(* Logix 5000 project; controller R5_CSS vendor 1 type 14 code 74 rev 19.11; software revision 19.01; part 16 of 20 *)
(* tags used below, declared in another part *)
   AlarmMaster : DINT;
   AllowHeatersWhenEmpty : BOOL;
   FT140_TOTAL_FLOW : REAL;
   HT_FAULT : BOOL;
   LC303B : LEVEL_CONTROL;   // INTERFACE LEVEL OF PRIMARY CONDENSER
   MV115B : ValveControl_TwoWay;
   MV301 : ValveControl_TwoWay;
   option_CartridgeHeaters : BOOL;
   P101A : PUMP_CONTROL;
   P101B : PUMP_CONTROL;
   P302A : PUMP_CONTROL;
   P302B : PUMP_CONTROL;
   P305 : PUMP_CONTROL;
   PID_JHE102 : PID;
   PID_JHE102_TON : TIMER;
   PID_TCV108 : PID;   // QUENCH FEED CONTROL VALVE
   PID_TCV108_Flow : PID;
   PID_TCV108_TON : TIMER;
   QuenchFlowMeterFailed : BOOL;
   QuenchTowerControlMode : BOOL;   // 0 = Temp.control 1 = Flow control
   TC101A : TEMP_CONTROL;   // QUENCH BASIN TRANSFER BASIN A TEMPERATURE CONTROL
   TC101B : TEMP_CONTROL;   // QUENCH BASIN TRANSFER BASIN B TEMPERATURE CONTROL
   TC108 : TEMP_CONTROL;   // QUENCH TOWER EXIT GAS TEMPERATURE CONTROL
   TC108_AUTO_ONS1 : BOOL;
   TC108_AUTO_ONS2 : BOOL;
   TC108_AutoStatic_SeekMaxSec : DINT;
   TC108_AutoStatic_SeekMaxTime : BOOL;
   TC108_AutoStatic_SeekMaxTmr : TIMER;
   TC108_AutoStatic_SeekTmr : TIMER;
   TC108_AutoStatic_SP : REAL;
   TC108_AutoStatic_SP_DB : REAL;
   TC108_AutoStatic_SP_DB_Down : REAL;
   TC108_AutoStatic_SP_DB_Up : REAL;
   TC108_manual_ONS1 : BOOL;
   TC108_QuenchFlowMeterFailedHold : REAL;
   TC108_QuenchFlowMeterFailedONS : BOOL;
   TC108_StaticMode : BOOL;
   TC108_StaticMode_Seek : BOOL;
   TC112 : TEMP_CONTROL;   // Quench Water Cartridge Heater ProcessTemp
   TC112_AUTO_Ons : BOOL;
   TC112_AUTO_Ons1 : BOOL;
   TC112_HeaterDisabled : BOOL;
   TC112_MANUAL_Ons : BOOL;
   TC112_NoPumpsRunningAlm : BOOL;
   TC112_START_TON : TIMER;
   TC112A : TEMP_CONTROL;
   TC313B : TEMP_CONTROL;   // PRIMARY COALESCER SHELL TEMPERATURE CONTROL
   TC319 : TEMP_CONTROL;   // COALESCER OIL CHAMBER PROCESS TEMPERATURE CONTROL
   TC319A : TEMP_CONTROL;   // COALESCER OIL CHAMBER SHEATH TEMPERATURE
   TMR_FAULT : DINT;
(* MainProgram, continued *)

ROUTINE TC101A_BasinPumpTemperature   (* ladder *)
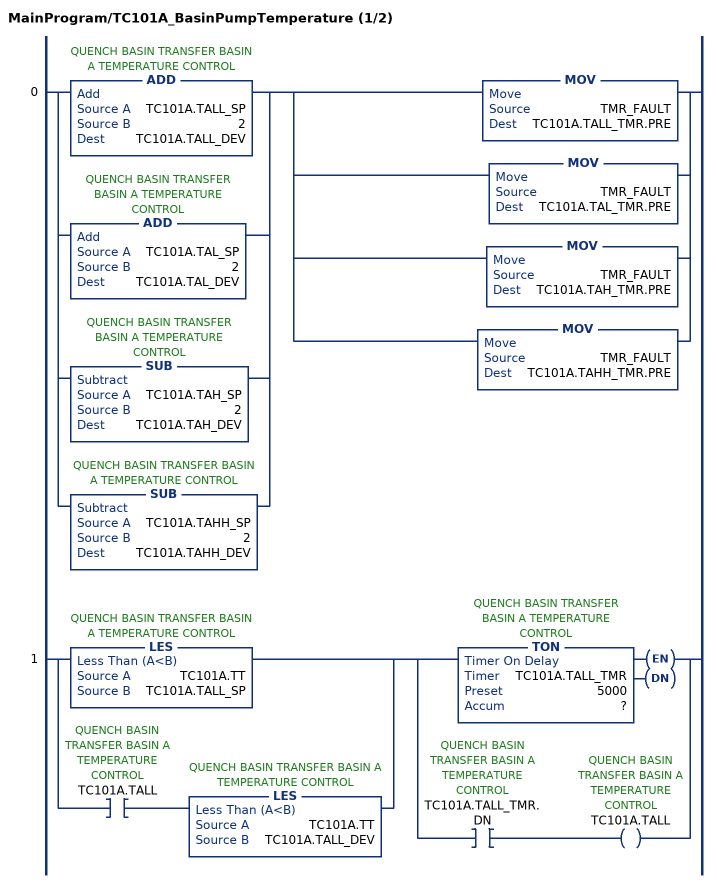
   0: [ADD(TC101A.TALL_SP,2,TC101A.TALL_DEV) ,ADD(TC101A.TAL_SP,2,TC101A.TAL_DEV) ,SUB(TC101A.TAH_SP,2,TC101A.TAH_DEV) ,SUB(TC101A.TAHH_SP,2,TC101A.TAHH_DEV) ][MOV(TMR_FAULT,TC101A.TALL_TMR.PRE) ,MOV(TMR_FAULT,TC101A.TAL_TMR.PRE) ,MOV(TMR_FAULT,TC101A.TAH_TMR.PRE) ,MOV(TMR_FAULT,TC101A.TAHH_TMR.PRE) ];
   1: [LES(TC101A.TT,TC101A.TALL_SP) ,XIC(TC101A.TALL) LES(TC101A.TT,TC101A.TALL_DEV) ][TON(TC101A.TALL_TMR,?,?) ,XIC(TC101A.TALL_TMR.DN) OTE(TC101A.TALL) ];
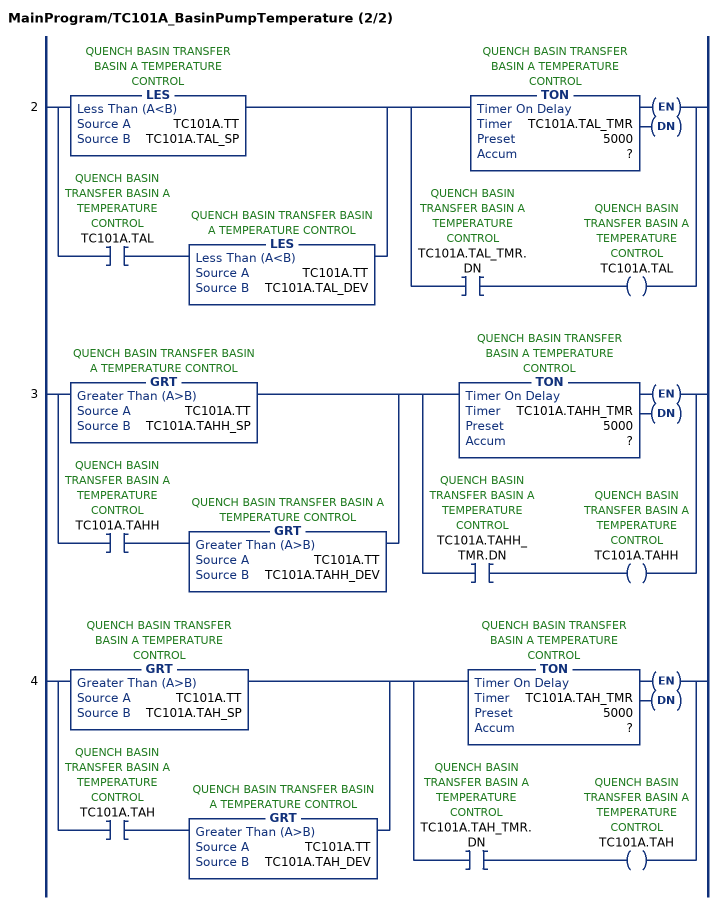
   2: [LES(TC101A.TT,TC101A.TAL_SP) ,XIC(TC101A.TAL) LES(TC101A.TT,TC101A.TAL_DEV) ][TON(TC101A.TAL_TMR,?,?) ,XIC(TC101A.TAL_TMR.DN) OTE(TC101A.TAL) ];
   3: [GRT(TC101A.TT,TC101A.TAHH_SP) ,XIC(TC101A.TAHH) GRT(TC101A.TT,TC101A.TAHH_DEV) ][TON(TC101A.TAHH_TMR,?,?) ,XIC(TC101A.TAHH_TMR.DN) OTE(TC101A.TAHH) ];
   4: [GRT(TC101A.TT,TC101A.TAH_SP) ,XIC(TC101A.TAH) GRT(TC101A.TT,TC101A.TAH_DEV) ][TON(TC101A.TAH_TMR,?,?) ,XIC(TC101A.TAH_TMR.DN) OTE(TC101A.TAH) ];
END_ROUTINE

ROUTINE TC101B_BasinPumpTemperature   (* ladder *)
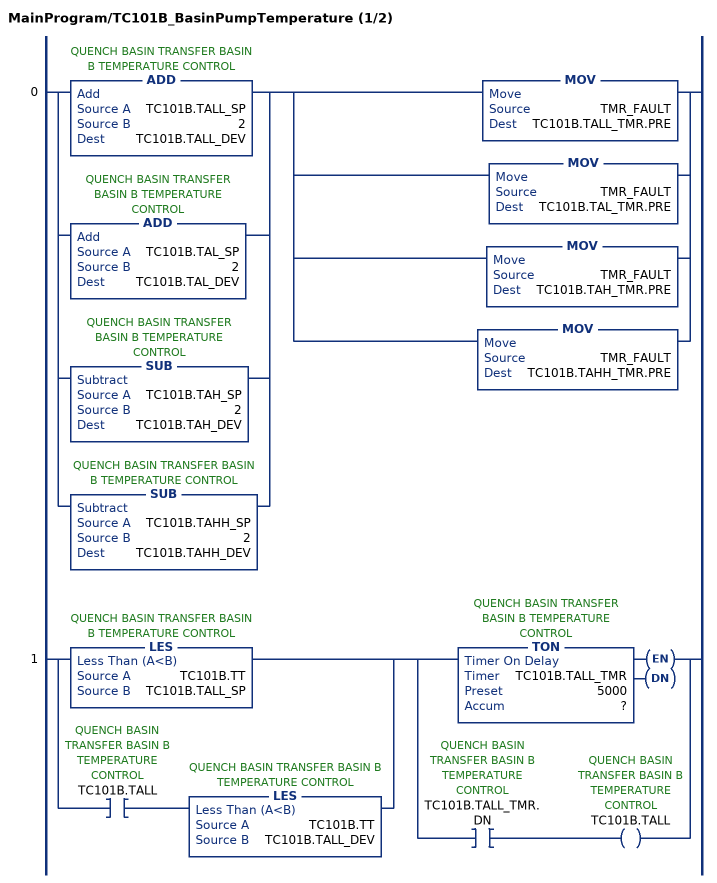
   0: [ADD(TC101B.TALL_SP,2,TC101B.TALL_DEV) ,ADD(TC101B.TAL_SP,2,TC101B.TAL_DEV) ,SUB(TC101B.TAH_SP,2,TC101B.TAH_DEV) ,SUB(TC101B.TAHH_SP,2,TC101B.TAHH_DEV) ][MOV(TMR_FAULT,TC101B.TALL_TMR.PRE) ,MOV(TMR_FAULT,TC101B.TAL_TMR.PRE) ,MOV(TMR_FAULT,TC101B.TAH_TMR.PRE) ,MOV(TMR_FAULT,TC101B.TAHH_TMR.PRE) ];
   1: [LES(TC101B.TT,TC101B.TALL_SP) ,XIC(TC101B.TALL) LES(TC101B.TT,TC101B.TALL_DEV) ][TON(TC101B.TALL_TMR,?,?) ,XIC(TC101B.TALL_TMR.DN) OTE(TC101B.TALL) ];
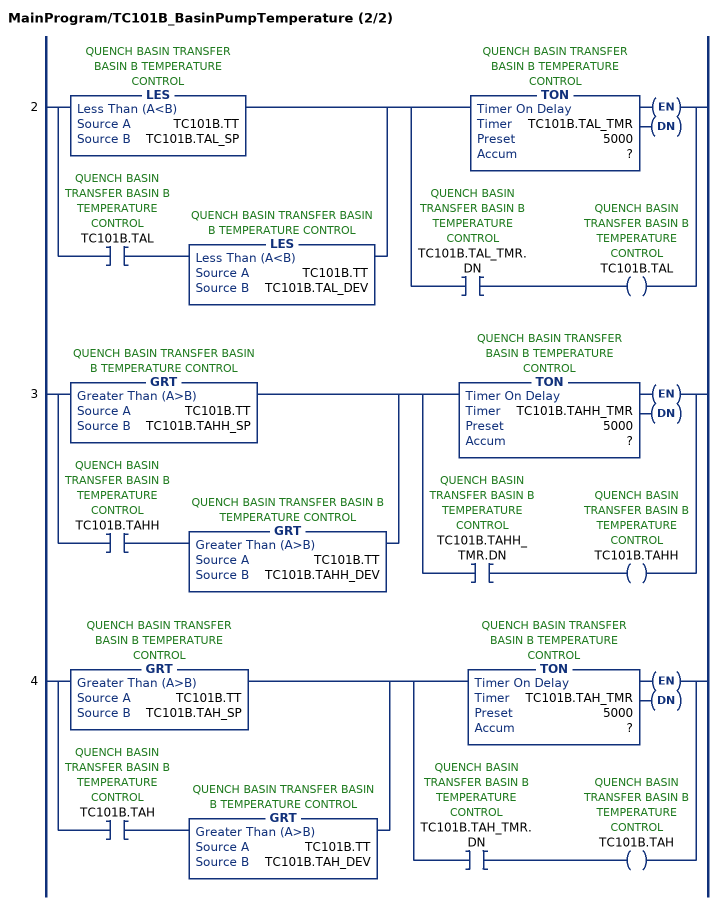
   2: [LES(TC101B.TT,TC101B.TAL_SP) ,XIC(TC101B.TAL) LES(TC101B.TT,TC101B.TAL_DEV) ][TON(TC101B.TAL_TMR,?,?) ,XIC(TC101B.TAL_TMR.DN) OTE(TC101B.TAL) ];
   3: [GRT(TC101B.TT,TC101B.TAHH_SP) ,XIC(TC101B.TAHH) GRT(TC101B.TT,TC101B.TAHH_DEV) ][TON(TC101B.TAHH_TMR,?,?) ,XIC(TC101B.TAHH_TMR.DN) OTE(TC101B.TAHH) ];
   4: [GRT(TC101B.TT,TC101B.TAH_SP) ,XIC(TC101B.TAH) GRT(TC101B.TT,TC101B.TAH_DEV) ][TON(TC101B.TAH_TMR,?,?) ,XIC(TC101B.TAH_TMR.DN) OTE(TC101B.TAH) ];
END_ROUTINE

ROUTINE TC108_QuenchTemperature_PID   (* ladder *)
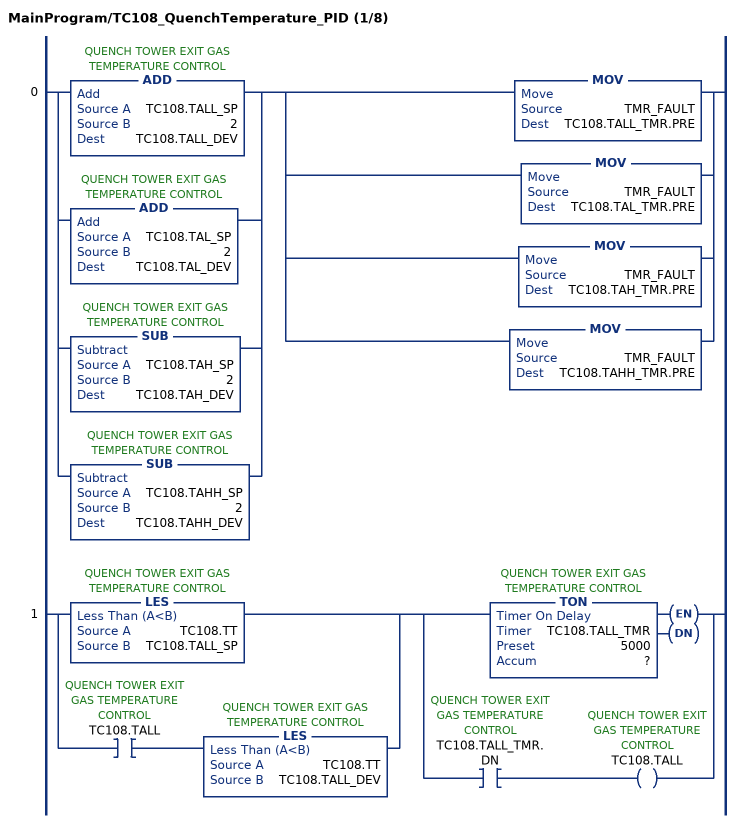
   0: [ADD(TC108.TALL_SP,2,TC108.TALL_DEV) ,ADD(TC108.TAL_SP,2,TC108.TAL_DEV) ,SUB(TC108.TAH_SP,2,TC108.TAH_DEV) ,SUB(TC108.TAHH_SP,2,TC108.TAHH_DEV) ][MOV(TMR_FAULT,TC108.TALL_TMR.PRE) ,MOV(TMR_FAULT,TC108.TAL_TMR.PRE) ,MOV(TMR_FAULT,TC108.TAH_TMR.PRE) ,MOV(TMR_FAULT,TC108.TAHH_TMR.PRE) ];
   1: [LES(TC108.TT,TC108.TALL_SP) ,XIC(TC108.TALL) LES(TC108.TT,TC108.TALL_DEV) ][TON(TC108.TALL_TMR,?,?) ,XIC(TC108.TALL_TMR.DN) OTE(TC108.TALL) ];
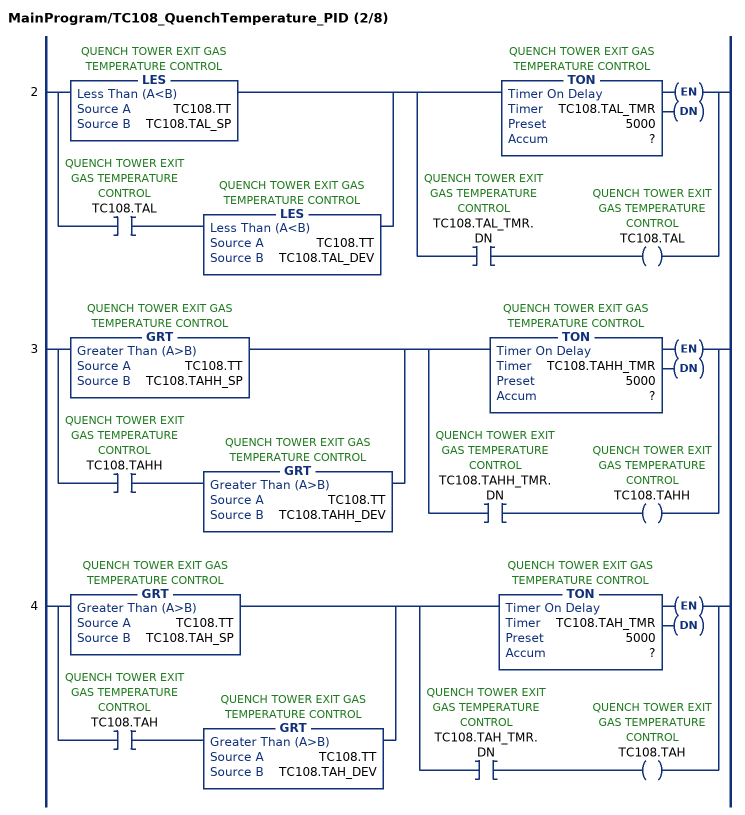
   2: [LES(TC108.TT,TC108.TAL_SP) ,XIC(TC108.TAL) LES(TC108.TT,TC108.TAL_DEV) ][TON(TC108.TAL_TMR,?,?) ,XIC(TC108.TAL_TMR.DN) OTE(TC108.TAL) ];
   3: [GRT(TC108.TT,TC108.TAHH_SP) ,XIC(TC108.TAHH) GRT(TC108.TT,TC108.TAHH_DEV) ][TON(TC108.TAHH_TMR,?,?) ,XIC(TC108.TAHH_TMR.DN) OTE(TC108.TAHH) ];
   4: [GRT(TC108.TT,TC108.TAH_SP) ,XIC(TC108.TAH) GRT(TC108.TT,TC108.TAH_DEV) ][TON(TC108.TAH_TMR,?,?) ,XIC(TC108.TAH_TMR.DN) OTE(TC108.TAH) ];
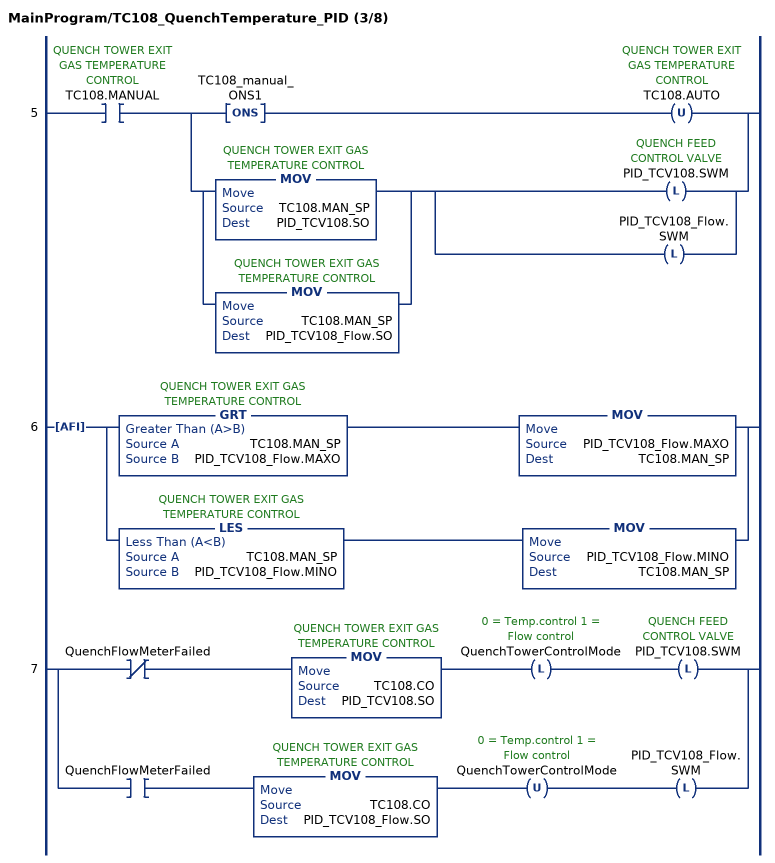
   5: XIC(TC108.MANUAL)[ONS(TC108_manual_ONS1) OTU(TC108.AUTO) ,[MOV(TC108.MAN_SP,PID_TCV108.SO) ,MOV(TC108.MAN_SP,PID_TCV108_Flow.SO) ] [OTL(PID_TCV108.SWM) ,OTL(PID_TCV108_Flow.SWM) ] ];
   6: AFI()[GRT(TC108.MAN_SP,PID_TCV108_Flow.MAXO) MOV(PID_TCV108_Flow.MAXO,TC108.MAN_SP) ,LES(TC108.MAN_SP,PID_TCV108_Flow.MINO) MOV(PID_TCV108_Flow.MINO,TC108.MAN_SP) ];
   7: [XIO(QuenchFlowMeterFailed) MOV(TC108.CO,PID_TCV108.SO) OTL(QuenchTowerControlMode) OTL(PID_TCV108.SWM) ,XIC(QuenchFlowMeterFailed) MOV(TC108.CO,PID_TCV108_Flow.SO) OTU(QuenchTowerControlMode) OTL(PID_TCV108_Flow.SWM) ];
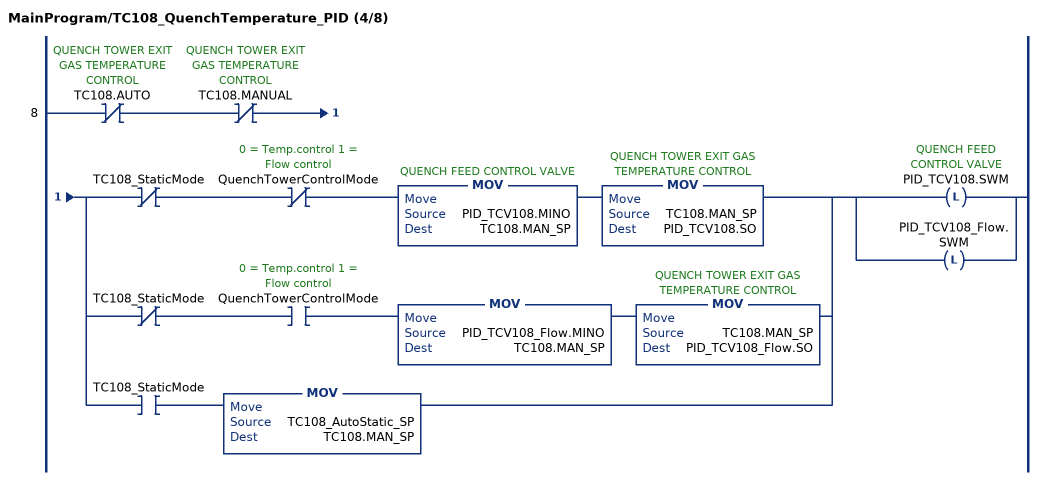
   8: XIO(TC108.AUTO)XIO(TC108.MANUAL)[XIO(TC108_StaticMode) XIO(QuenchTowerControlMode) MOV(PID_TCV108.MINO,TC108.MAN_SP) MOV(TC108.MAN_SP,PID_TCV108.SO) ,XIO(TC108_StaticMode) XIC(QuenchTowerControlMode) MOV(PID_TCV108_Flow.MINO,TC108.MAN_SP) MOV(TC108.MAN_SP,PID_TCV108_Flow.SO) ,XIC(TC108_StaticMode) MOV(TC108_AutoStatic_SP,TC108.MAN_SP) ][OTL(PID_TCV108.SWM) ,OTL(PID_TCV108_Flow.SWM) ];
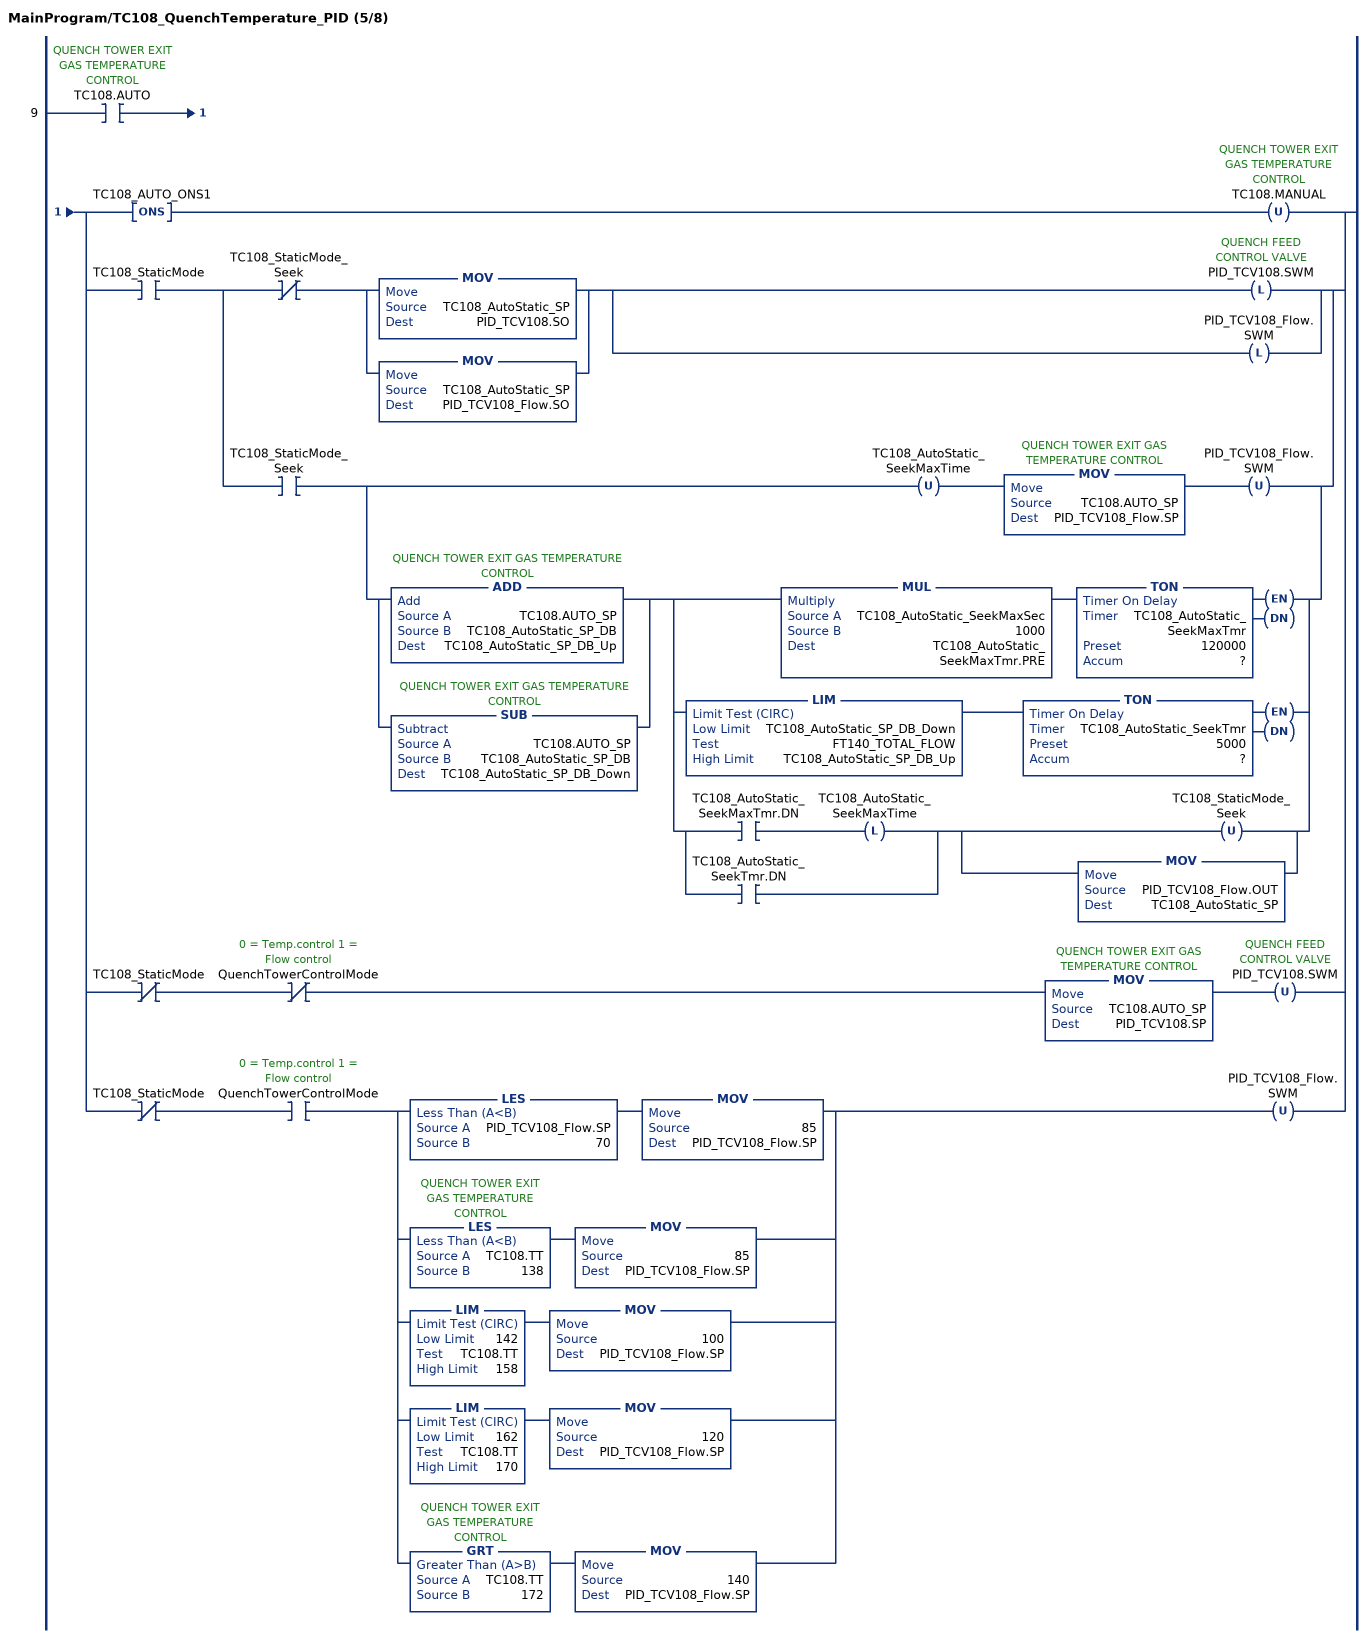
   9: XIC(TC108.AUTO)[ONS(TC108_AUTO_ONS1) OTU(TC108.MANUAL) ,XIC(TC108_StaticMode) [XIO(TC108_StaticMode_Seek) [MOV(TC108_AutoStatic_SP,PID_TCV108.SO) ,MOV(TC108_AutoStatic_SP,PID_TCV108_Flow.SO) ] [OTL(PID_TCV108.SWM) ,OTL(PID_TCV108_Flow.SWM) ] ,XIC(TC108_StaticMode_Seek) [OTU(TC108_AutoStatic_SeekMaxTime) MOV(TC108.AUTO_SP,PID_TCV108_Flow.SP) OTU(PID_TCV108_Flow.SWM) ,[ADD(TC108.AUTO_SP,TC108_AutoStatic_SP_DB,TC108_AutoStatic_SP_DB_Up) ,SUB(TC108.AUTO_SP,TC108_AutoStatic_SP_DB,TC108_AutoStatic_SP_DB_Down) ] [MUL(TC108_AutoStatic_SeekMaxSec,1000,TC108_AutoStatic_SeekMaxTmr.PRE) TON(TC108_AutoStatic_SeekMaxTmr,?,?) ,LIM(TC108_AutoStatic_SP_DB_Down,FT140_TOTAL_FLOW,TC108_AutoStatic_SP_DB_Up) TON(TC108_AutoStatic_SeekTmr,?,?) ,[XIC(TC108_AutoStatic_SeekMaxTmr.DN) OTL(TC108_AutoStatic_SeekMaxTime) ,XIC(TC108_AutoStatic_SeekTmr.DN) ] [OTU(TC108_StaticMode_Seek) ,MOV(PID_TCV108_Flow.OUT,TC108_AutoStatic_SP) ] ] ] ] ,XIO(TC108_StaticMode) XIO(QuenchTowerControlMode) MOV(TC108.AUTO_SP,PID_TCV108.SP) OTU(PID_TCV108.SWM) ,XIO(TC108_StaticMode) XIC(QuenchTowerControlMode) [LES(PID_TCV108_Flow.SP,70) MOV(85,PID_TCV108_Flow.SP) ,LES(TC108.TT,138) MOV(85,PID_TCV108_Flow.SP) ,LIM(142,TC108.TT,158) MOV(100,PID_TCV108_Flow.SP) ,LIM(162,TC108.TT,170) MOV(120,PID_TCV108_Flow.SP) ,GRT(TC108.TT,172) MOV(140,PID_TCV108_Flow.SP) ] OTU(PID_TCV108_Flow.SWM) ];
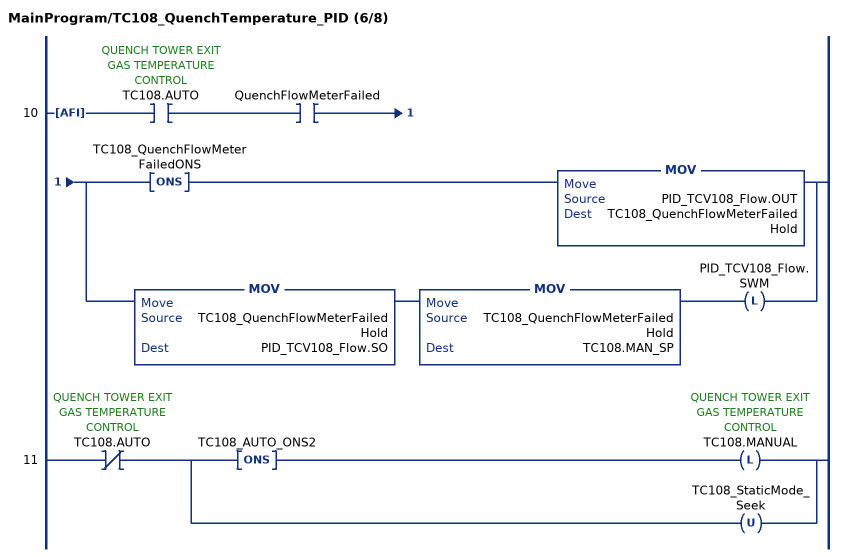
   10: AFI()XIC(TC108.AUTO)XIC(QuenchFlowMeterFailed)[ONS(TC108_QuenchFlowMeterFailedONS) MOV(PID_TCV108_Flow.OUT,TC108_QuenchFlowMeterFailedHold) ,MOV(TC108_QuenchFlowMeterFailedHold,PID_TCV108_Flow.SO) MOV(TC108_QuenchFlowMeterFailedHold,TC108.MAN_SP) OTL(PID_TCV108_Flow.SWM) ];
   11: XIO(TC108.AUTO)[ONS(TC108_AUTO_ONS2) OTL(TC108.MANUAL) ,OTU(TC108_StaticMode_Seek) ];
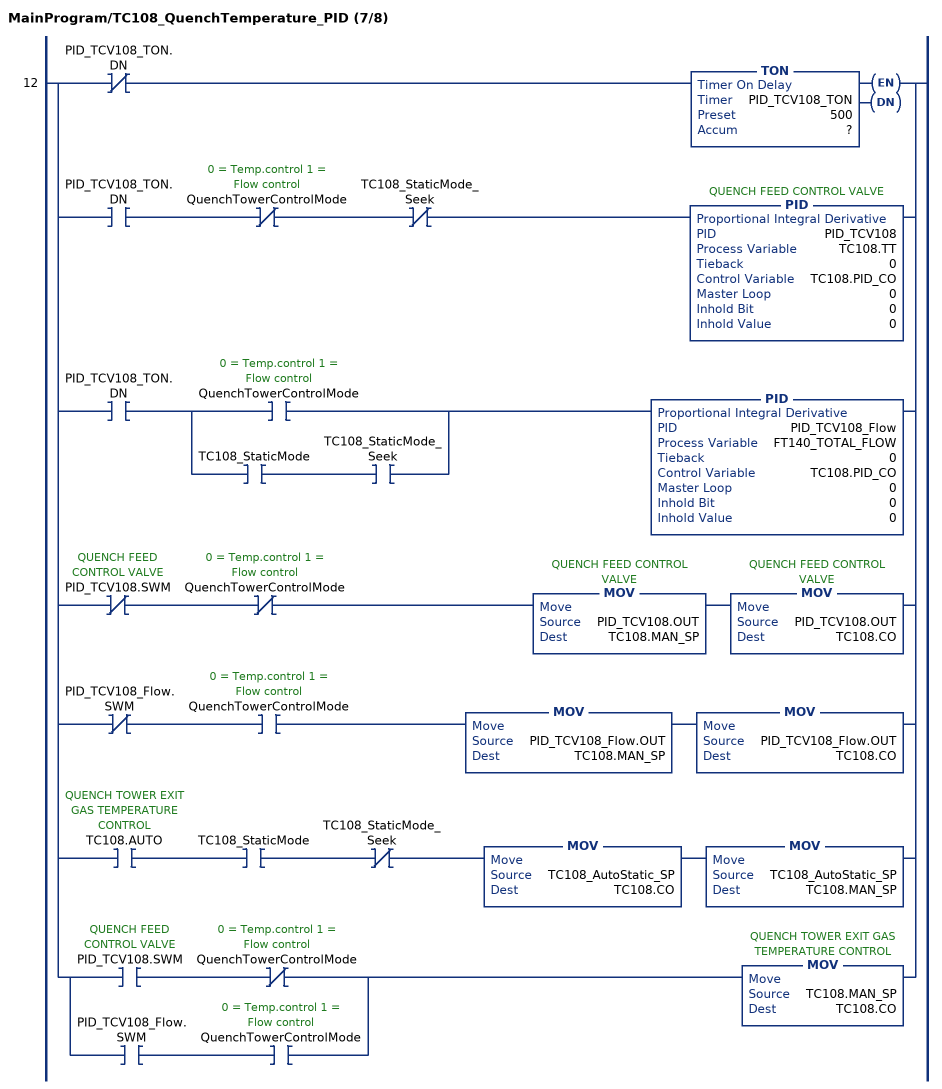
   12: [XIO(PID_TCV108_TON.DN) TON(PID_TCV108_TON,?,?) ,XIC(PID_TCV108_TON.DN) XIO(QuenchTowerControlMode) XIO(TC108_StaticMode_Seek) PID(PID_TCV108,TC108.TT,0,TC108.PID_CO,0,0,0) ,XIC(PID_TCV108_TON.DN) [XIC(QuenchTowerControlMode) ,XIC(TC108_StaticMode) XIC(TC108_StaticMode_Seek) ] PID(PID_TCV108_Flow,FT140_TOTAL_FLOW,0,TC108.PID_CO,0,0,0) ,XIO(PID_TCV108.SWM) XIO(QuenchTowerControlMode) MOV(PID_TCV108.OUT,TC108.MAN_SP) MOV(PID_TCV108.OUT,TC108.CO) ,XIO(PID_TCV108_Flow.SWM) XIC(QuenchTowerControlMode) MOV(PID_TCV108_Flow.OUT,TC108.MAN_SP) MOV(PID_TCV108_Flow.OUT,TC108.CO) ,XIC(TC108.AUTO) XIC(TC108_StaticMode) XIO(TC108_StaticMode_Seek) MOV(TC108_AutoStatic_SP,TC108.CO) MOV(TC108_AutoStatic_SP,TC108.MAN_SP) ,[XIC(PID_TCV108.SWM) XIO(QuenchTowerControlMode) ,XIC(PID_TCV108_Flow.SWM) XIC(QuenchTowerControlMode) ] MOV(TC108.MAN_SP,TC108.CO) ];
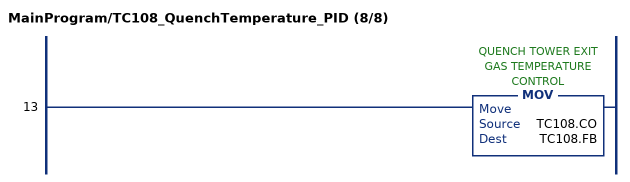
   13: MOV(TC108.CO,TC108.FB);
END_ROUTINE

ROUTINE TC112_CoalWaterTempHeater_PID   (* ladder *)
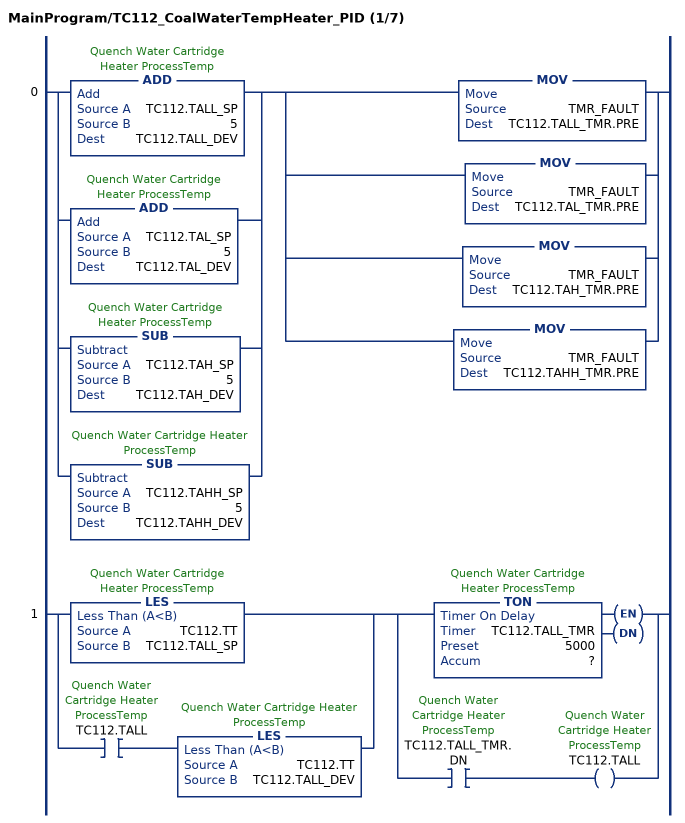
   0: [ADD(TC112.TALL_SP,5,TC112.TALL_DEV) ,ADD(TC112.TAL_SP,5,TC112.TAL_DEV) ,SUB(TC112.TAH_SP,5,TC112.TAH_DEV) ,SUB(TC112.TAHH_SP,5,TC112.TAHH_DEV) ][MOV(TMR_FAULT,TC112.TALL_TMR.PRE) ,MOV(TMR_FAULT,TC112.TAL_TMR.PRE) ,MOV(TMR_FAULT,TC112.TAH_TMR.PRE) ,MOV(TMR_FAULT,TC112.TAHH_TMR.PRE) ];
   1: [LES(TC112.TT,TC112.TALL_SP) ,XIC(TC112.TALL) LES(TC112.TT,TC112.TALL_DEV) ][TON(TC112.TALL_TMR,?,?) ,XIC(TC112.TALL_TMR.DN) OTE(TC112.TALL) ];
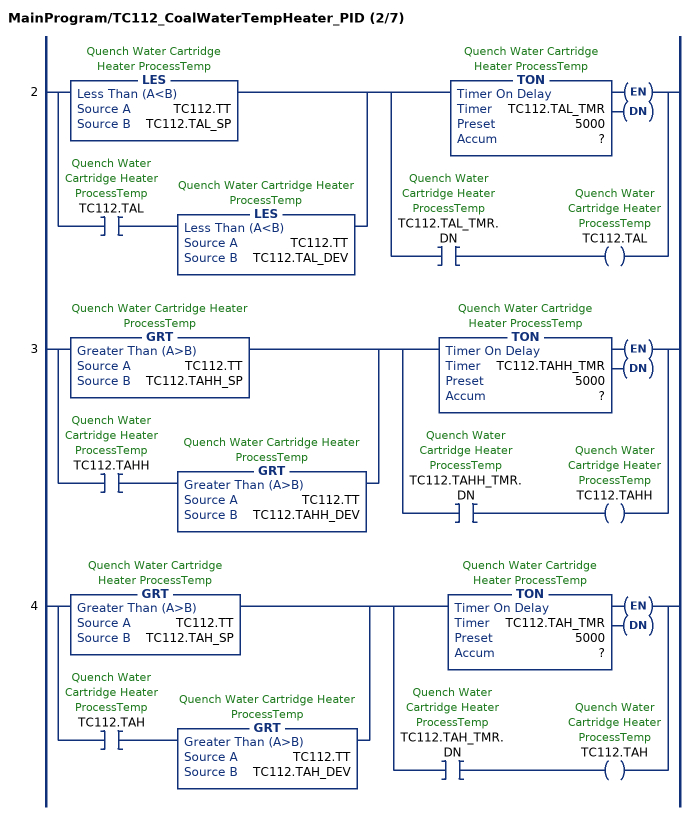
   2: [LES(TC112.TT,TC112.TAL_SP) ,XIC(TC112.TAL) LES(TC112.TT,TC112.TAL_DEV) ][TON(TC112.TAL_TMR,?,?) ,XIC(TC112.TAL_TMR.DN) OTE(TC112.TAL) ];
   3: [GRT(TC112.TT,TC112.TAHH_SP) ,XIC(TC112.TAHH) GRT(TC112.TT,TC112.TAHH_DEV) ][TON(TC112.TAHH_TMR,?,?) ,XIC(TC112.TAHH_TMR.DN) OTE(TC112.TAHH) ];
   4: [GRT(TC112.TT,TC112.TAH_SP) ,XIC(TC112.TAH) GRT(TC112.TT,TC112.TAH_DEV) ][TON(TC112.TAH_TMR,?,?) ,XIC(TC112.TAH_TMR.DN) OTE(TC112.TAH) ];
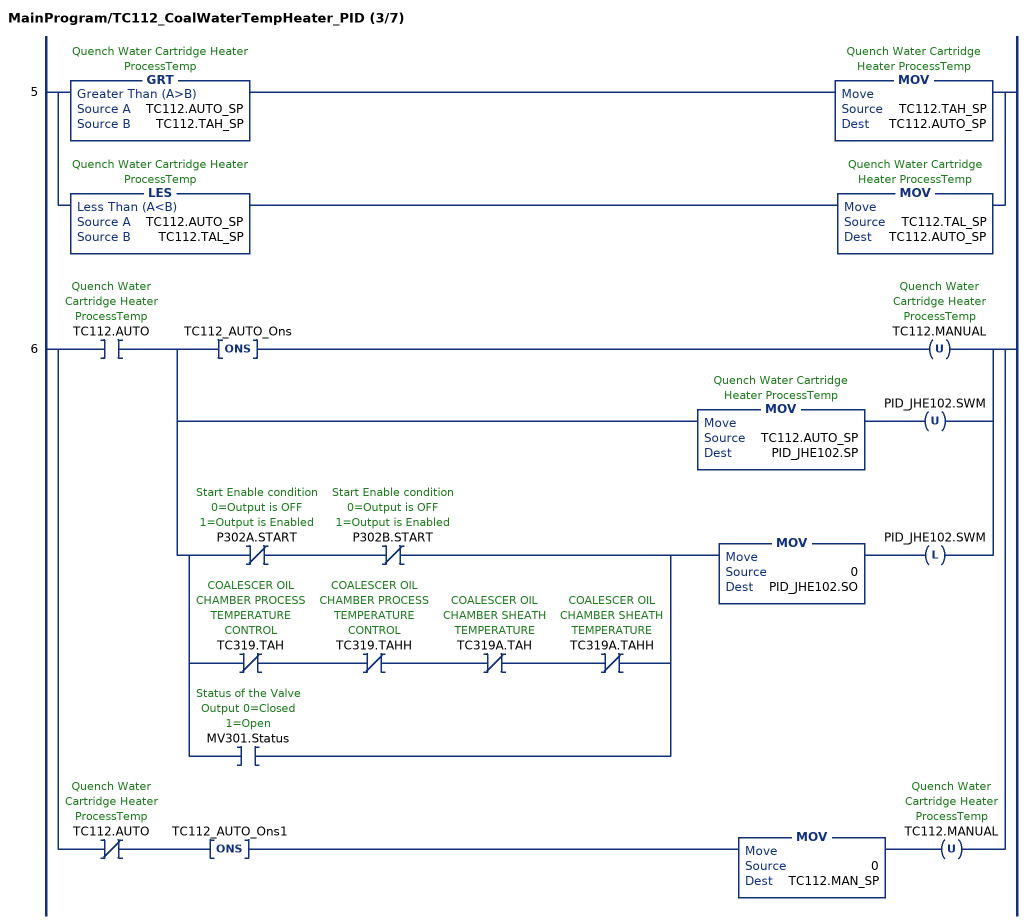
   5: [GRT(TC112.AUTO_SP,TC112.TAH_SP) MOV(TC112.TAH_SP,TC112.AUTO_SP) ,LES(TC112.AUTO_SP,TC112.TAL_SP) MOV(TC112.TAL_SP,TC112.AUTO_SP) ];
   6: [XIC(TC112.AUTO) [ONS(TC112_AUTO_Ons) OTU(TC112.MANUAL) ,MOV(TC112.AUTO_SP,PID_JHE102.SP) OTU(PID_JHE102.SWM) ,[XIO(P302A.START) XIO(P302B.START) ,XIO(TC319.TAH) XIO(TC319.TAHH) XIO(TC319A.TAH) XIO(TC319A.TAHH) ,XIC(MV301.Status) ] MOV(0,PID_JHE102.SO) OTL(PID_JHE102.SWM) ] ,XIO(TC112.AUTO) ONS(TC112_AUTO_Ons1) MOV(0,TC112.MAN_SP) OTU(TC112.MANUAL) ];
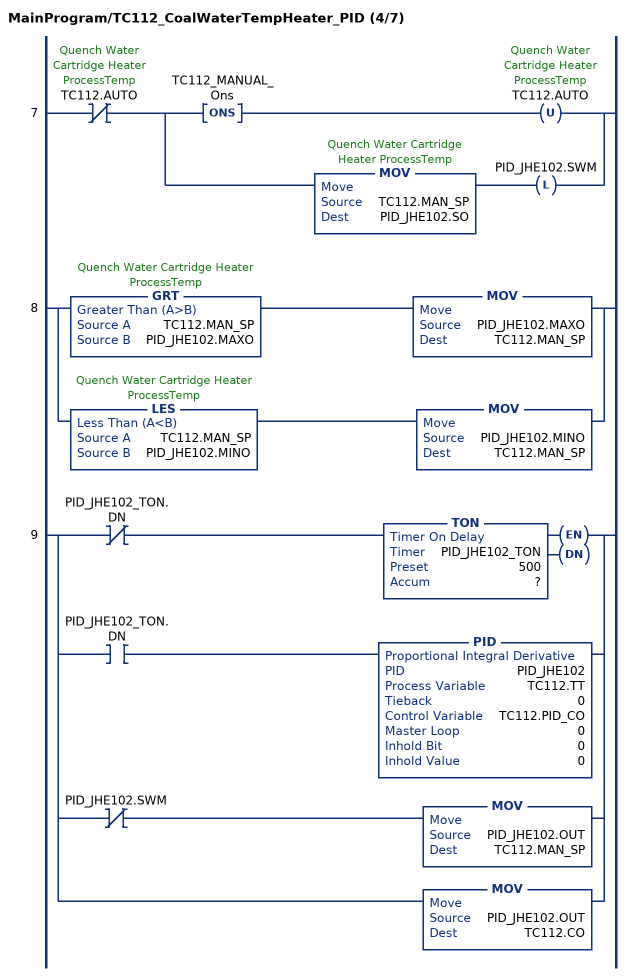
   7: XIO(TC112.AUTO)[ONS(TC112_MANUAL_Ons) OTU(TC112.AUTO) ,MOV(TC112.MAN_SP,PID_JHE102.SO) OTL(PID_JHE102.SWM) ];
   8: [GRT(TC112.MAN_SP,PID_JHE102.MAXO) MOV(PID_JHE102.MAXO,TC112.MAN_SP) ,LES(TC112.MAN_SP,PID_JHE102.MINO) MOV(PID_JHE102.MINO,TC112.MAN_SP) ];
   9: [XIO(PID_JHE102_TON.DN) TON(PID_JHE102_TON,?,?) ,XIC(PID_JHE102_TON.DN) PID(PID_JHE102,TC112.TT,0,TC112.PID_CO,0,0,0) ,XIO(PID_JHE102.SWM) MOV(PID_JHE102.OUT,TC112.MAN_SP) ,MOV(PID_JHE102.OUT,TC112.CO) ];
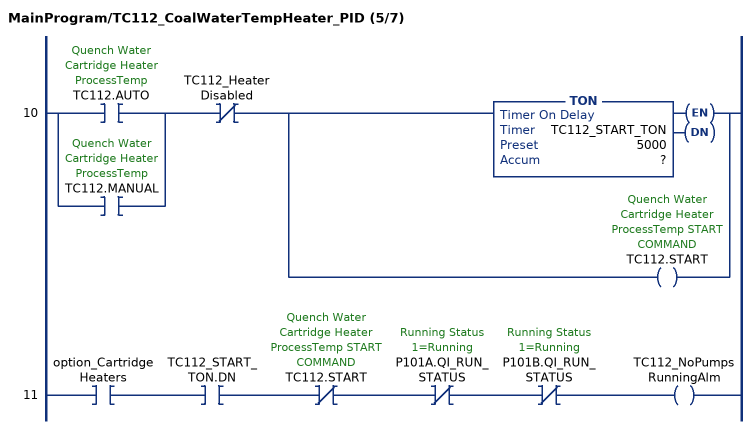
   10: [XIC(TC112.AUTO) ,XIC(TC112.MANUAL) ]XIO(TC112_HeaterDisabled)[TON(TC112_START_TON,?,?) ,OTE(TC112.START) ];
   11: XIC(option_CartridgeHeaters)XIC(TC112_START_TON.DN)XIO(TC112.START)XIO(P101A.QI_RUN_STATUS)XIO(P101B.QI_RUN_STATUS)OTE(TC112_NoPumpsRunningAlm);
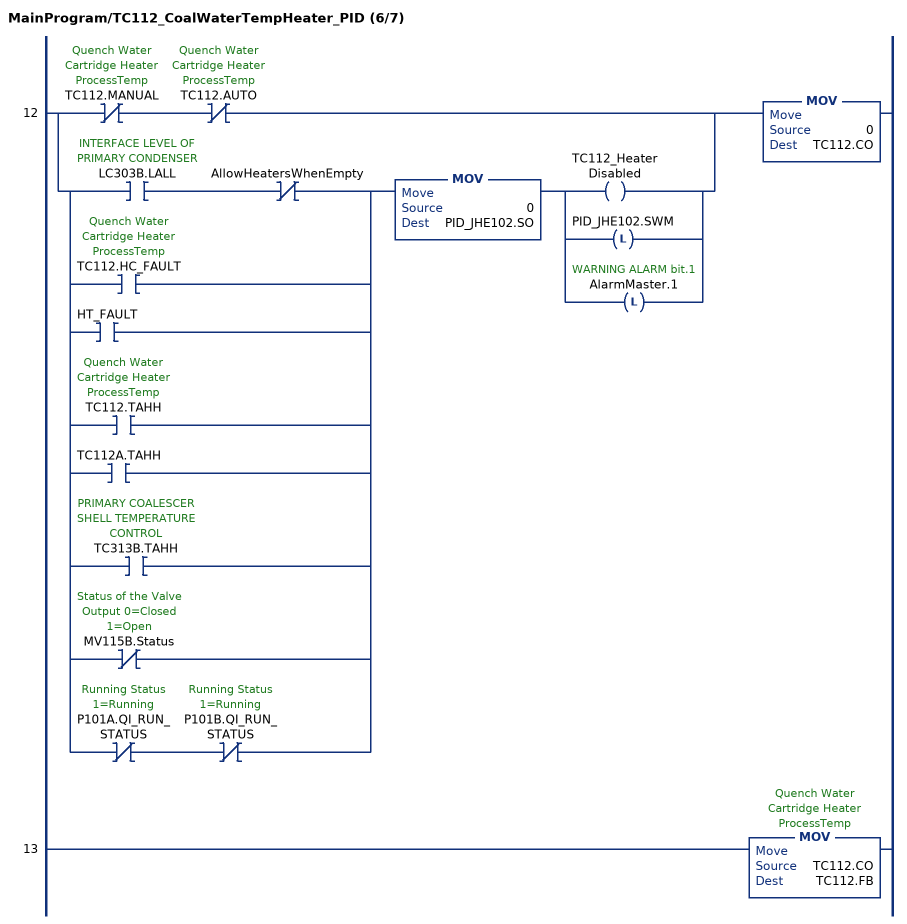
   12: [XIO(TC112.MANUAL) XIO(TC112.AUTO) ,[XIC(LC303B.LALL) XIO(AllowHeatersWhenEmpty) ,XIC(TC112.HC_FAULT) ,XIC(HT_FAULT) ,XIC(TC112.TAHH) ,XIC(TC112A.TAHH) ,XIC(TC313B.TAHH) ,XIO(MV115B.Status) ,XIO(P101A.QI_RUN_STATUS) XIO(P101B.QI_RUN_STATUS) ] MOV(0,PID_JHE102.SO) [OTE(TC112_HeaterDisabled) ,OTL(PID_JHE102.SWM) ,OTL(AlarmMaster.1) ] ]MOV(0,TC112.CO);
   13: MOV(TC112.CO,TC112.FB);
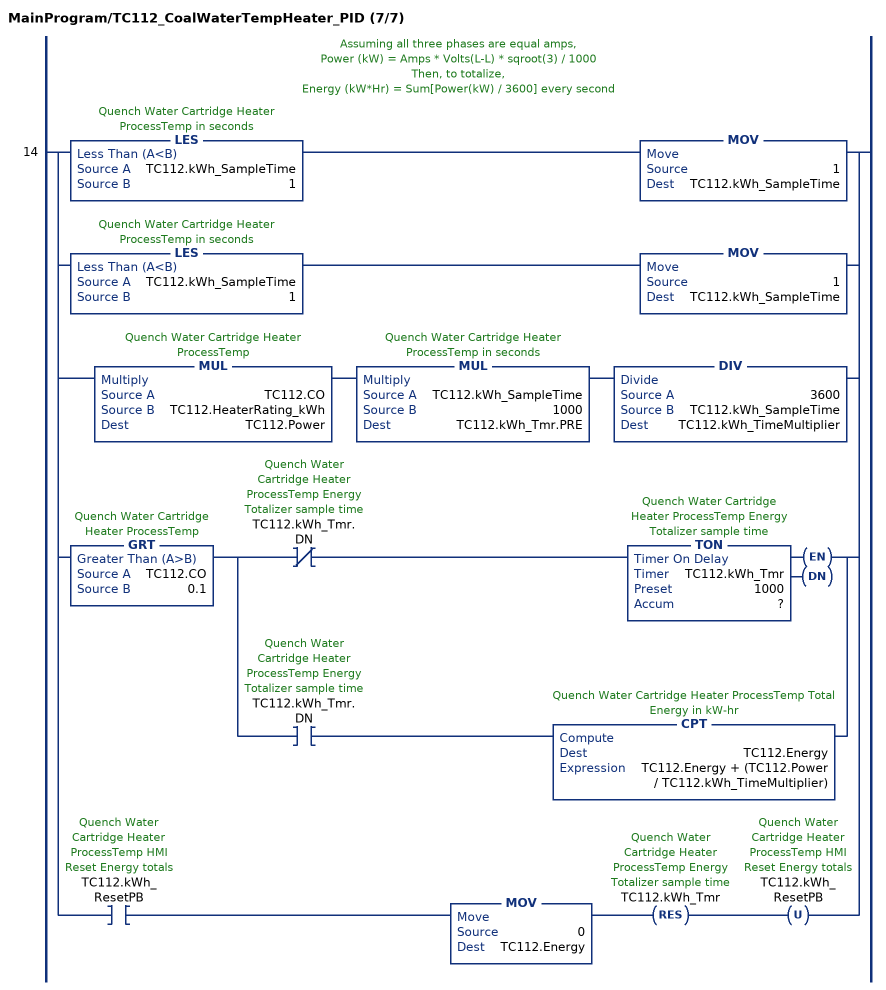
   // Assuming all three phases are equal amps,
   // Power (kW) = Amps * Volts(L-L) * sqroot(3) / 1000
   // Then, to totalize,
   // Energy (kW*Hr) = Sum[Power(kW) / 3600] every second
   14: [[LES(TC112.kWh_SampleTime,1) MOV(1,TC112.kWh_SampleTime) ,LES(TC112.kWh_SampleTime,1) MOV(1,TC112.kWh_SampleTime) ] ,MUL(TC112.CO,TC112.HeaterRating_kWh,TC112.Power) MUL(TC112.kWh_SampleTime,1000,TC112.kWh_Tmr.PRE) DIV(3600,TC112.kWh_SampleTime,TC112.kWh_TimeMultiplier) ,GRT(TC112.CO,0.1) [XIO(TC112.kWh_Tmr.DN) TON(TC112.kWh_Tmr,?,?) ,XIC(TC112.kWh_Tmr.DN) CPT(TC112.Energy,TC112.Energy + (TC112.Power / TC112.kWh_TimeMultiplier)) ] ,XIC(TC112.kWh_ResetPB) MOV(0,TC112.Energy) RES(TC112.kWh_Tmr) OTU(TC112.kWh_ResetPB) ];
END_ROUTINE
